FUNCTION_BLOCK SuppressPuls (* Composite Function Block Type *)
  (* Standard: 61499-2 *)
  (* Version 0.0, 6/2/2026, Schneider Electric, template *)
  PACKAGE SE.Nereda;
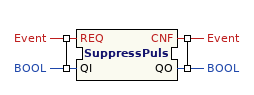
  EVENT_INPUT
    REQ WITH QI; (* Normal Execution Request *)
  END_EVENT
  EVENT_OUTPUT
    CNF WITH QO; (* Execution Confirmation *)
  END_EVENT
  VAR_INPUT
    QI : BOOL; (* Input event qualifier *)
  END_VAR
  VAR_OUTPUT
    QO : BOOL; (* Output event qualifier *)
  END_VAR
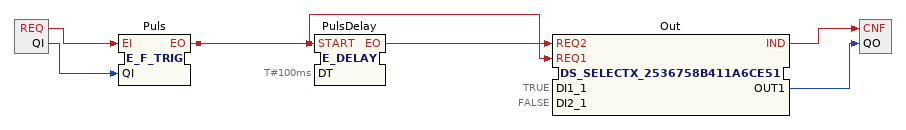
  FBS
    Puls : E_F_TRIG;
    PulsDelay : E_DELAY(DT := T#100ms);
    Out : DS_SELECTX_2536758B411A6CE51(DI1_1 := TRUE, DI2_1 := FALSE); {SET_ATTRIBUTE(Configuration.GenericFBType.InterfaceParams, Runtime.Standard#CNTX:=2;CNTY:=1;DI${CNTX,_,CNTY$}:BOOL)}
  END_FBS
  EVENT_CONNECTIONS
    REQ TO Puls.EI;
    Puls.EO TO PulsDelay.START;
    Out.IND TO CNF;
    PulsDelay.EO TO Out.REQ2;
    Puls.EO TO Out.REQ1;
  END_CONNECTIONS
  DATA_CONNECTIONS
    QI TO Puls.QI;
    Out.OUT1 TO QO;
  END_CONNECTIONS
END_FUNCTION_BLOCK
